FUNCTION_BLOCK FB_PartStation EXTENDS FB_Module IMPLEMENTS I_GantryPart
VAR_INPUT
	Axis				: REFERENCE TO AXIS_REF;
	ipGantry			: I_GantryPart;
	cmd					: E_PartStationCommand := E_PartStationCommand.None;
	
	inpSim				: BOOL := TRUE;
	inpPartPresent		AT %I* : BOOL;
END_VAR
VAR_OUTPUT
	stsState			: E_PartStationState := E_PartStationState.Idle;
	stsCurrentStep		: DINT;
END_VAR
VAR
	//Devices
	Conveyor			: FB_Axis;
	
	DebounceTimer		: TON;
	DebounceTime		: TIME := T#500MS;
	PP_DepartSimTimer	: TON;
	PP_ArriveSimTimer	: TON;
	
	rtStarting			: R_TRIG;
	rtStopping			: R_TRIG;
	rtPartPresent		: R_TRIG;

	GantryClear			: BOOL;
	GantryPickComplete	: BOOL;
END_VAR

Map();
Status();
StateMachine();

METHOD Aborting : BOOL
VAR_INPUT
END_VAR
Conveyor.cmd := E_AxisCommand.Stop;
stsCurrentStep := 0;
END_METHOD

METHOD Map : BOOL
VAR_INPUT
END_VAR
Conveyor(Axis := Axis);

DebounceTimer(IN := inpPartPresent, PT := DebounceTime);

GantryClear := ipGantry.PartReady;
GantryPickComplete := ipGantry.PartPicked;
END_METHOD

{warning 'add property implementation'}
PROPERTY PartPicked : BOOL
GET
PartPicked := NOT inpPartPresent;
END_GET
END_PROPERTY

{warning 'add property implementation'}
PROPERTY PartReady : BOOL
GET
PartReady := inpPartPresent AND Conveyor.stsVelocity = 0;
END_GET
END_PROPERTY

METHOD Simulate : BOOL
VAR_INPUT
END_VAR
rtPartPresent(CLK := GantryPickComplete);
inpPartPresent R= rtPartPresent.Q;

PP_ArriveSimTimer(IN := stsState = E_PartStationState.Running AND NOT inpPartPresent, PT := T#5S);
inpPartPresent S= PP_ArriveSimTimer.Q;
END_METHOD

METHOD Starting : BOOL
VAR_INPUT
END_VAR
CASE stsCurrentStep OF
	1000: //Turn on conveyor servo
		Conveyor.cmd := E_AxisCommand.TurnOn;
		IF Conveyor.stsState = E_AxisState.Ready THEN
			stsCurrentStep := 1010;
		END_IF
	1010: //Start conveyor at 100 mm/s (arbitrary value)
		Conveyor.inpVelocity := 100;
		Conveyor.cmd := E_AxisCommand.ExecuteMoveVel;
		IF Conveyor.stsVelocity > 0 THEN
			stsCurrentStep := 0;
		END_IF
END_CASE
END_METHOD

METHOD StateMachine : BOOL
VAR_INPUT
END_VAR
IF inpSim THEN
	Simulate();
END_IF

CASE stsState OF
	E_PartStationState.Idle: //Station is idle and ready for command
		IF cmd = E_PartStationCommand.Start THEN
			stsState := E_PartStationState.Starting;
		END_IF
	E_PartStationState.Starting: //Start conveyor and ready for parts
		Starting();
		IF stsCurrentStep = 0 AND Conveyor.stsVelocity > 0 THEN
			stsState := E_PartStationState.Running;
		END_IF
	E_PartStationState.Running: //Running and waiting for part present sensor
		IF DebounceTimer.Q THEN
			Stopping();
			stsState := E_PartStationState.Stopping;
		END_IF
	E_PartStationState.Stopping: //Stopping conveyor
		Stopping();
		IF stsCurrentStep = 0 AND Conveyor.stsVelocity = 0 THEN
			stsState := E_PartStationState.Stopped;
		END_IF
	E_PartStationState.Stopped: //Conveyor stopped. waiting for part pick
		IF NOT inpPartPresent AND GantryClear THEN
			Starting();
			stsState := E_PartStationState.Starting;
		END_IF
	E_PartStationState.Aborting: //Abort all station activity
		Aborting();
		IF stsCurrentStep = 0 AND Conveyor.stsVelocity = 0 THEN
			stsState := E_PartStationState.Idle;
		END_IF
END_CASE

IF cmd = E_PartStationCommand.Abort THEN
	stsState := E_PartStationState.Aborting;
END_IF

cmd := E_PartStationCommand.None;
END_METHOD

METHOD Status : BOOL
VAR_INPUT
END_VAR
//State transition one shots
rtStarting(CLK := stsState = E_PalletStationState.Starting);
IF rtStarting.Q THEN
	stsCurrentStep := 1000;
END_IF

rtStopping(CLK := stsState = E_PartStationState.Stopping);
IF rtStopping.Q THEN
	stsCurrentStep := 2000;
END_IF
END_METHOD

METHOD Stopping : BOOL
VAR_INPUT
END_VAR

VAR
	END_IFCASE: INT;
END_VAR
CASE stsCurrentStep OF
	2000: //Stop conveyor
		Conveyor.cmd := E_AxisCommand.Stop;
		IF Conveyor.stsVelocity = 0 THEN
			stsCurrentStep := 0;
		END_IF
END_CASE
END_METHOD

END_FUNCTION_BLOCK

(* stored: Version 1.1.0.1, ProductVersion 3.1.4024.4
   POU FB_PartStation: Id {21b06fcb-7bab-4e72-a22c-2c772da71df6}, SpecialFunc None
   Method Aborting: Id {d32ecc30-a2d1-4b92-b962-d7113a4121fc}
   Method Map: Id {55f3ddf8-6288-45e8-9b4b-1816ca7aeda6}
   Property PartPicked: Id {e872d0a9-9f22-470e-b8ca-d0cd5c4cc9e3}
   Get Get: Id {f5d103e5-a2a9-4368-abf3-2ba4a3438f1a}
   Property PartReady: Id {4c6a83d0-09fe-46a4-bcf8-e3248f24f1d6}
   Get Get: Id {00d02a12-e6f3-4898-89f4-1c9cdfc5c0ee}
   Method Simulate: Id {d878782c-2bce-4eb5-a19f-b52546e65167}
   Method Starting: Id {89881208-c2af-4fe6-9318-93a8965acadf}
   Method StateMachine: Id {40d31a89-e600-4fb9-8580-b0e24ab4d585}
   Method Status: Id {1fe6d3c7-7eba-4770-861a-340f536e11cb}
   Method Stopping: Id {d03b5ad8-5f22-479e-95d5-240a584b2e54} *)
